// A sink that was never part of a run writes nothing.
//
// The distinction is RunStarted. Without it no document was ever opened, so there
// is nothing to write and inventing one would claim something happened.
//
// AN EMPTY RUN IS DIFFERENT and does produce a document, carrying tests="0" - the
// second half of this test. That is the reverse of the behaviour before RunStarted
// existed, and deliberately so: a missing file is ambiguous, because a
// configuration problem and a run with no tests look identical from CI. R3 one
// level up.
FUNCTION_BLOCK TEST_JUnitReporterWritesNothingWhenNothingRan IMPLEMENTS I_Test
VAR
	Writer : TestJUnitReporter;
	Spy	   : SpyReporter;
	Tally  : TestRunTally;
	Phase  : DINT;
	Scans  : DINT;
	Path : T_MaxString := 'C:\ProgramData\Beckhoff\TwinCAT\3.1\Boot\TestHarnessCoreVerifier_Empty.xml';
	ExpectedCount : UDINT;
	ActualCount	  : UDINT;
END_VAR

METHOD Run : BOOL
VAR_INPUT
	Enable : BOOL;
	Test   : I_TestAssertions;
END_VAR
Scans := Scans + 1;
IF Scans > 2000 THEN
	Test.Fail('the write never finished');
	Run := TRUE;
	RETURN;
END_IF

CASE Phase OF

0:
	Writer.SetPath(Path);
	Writer.AttachErrorSink(Spy);

	// No RunStarted either, so no document is ever opened.
	Tally.SetLabel('nothing');
	Tally.Begin(0);
	Tally.Finish();
	Writer.RunFinished(Status := Tally, TargetInfo := 'the verifier');
	Phase := 1;
	Run	  := FALSE;

1:
	Test.AssertTrue(Writer.IsIdle, 'no write was started');

	ExpectedCount := 0;
	ActualCount	  := Writer.FilesWritten;
	Test.AssertEqual(ExpectedCount, ActualCount, 'nothing was written');

	// Not an error either - an empty run is a legitimate deployment.
	ActualCount := Writer.WriteFailures;
	Test.AssertEqual(ExpectedCount, ActualCount, 'and that is not a failure');

	ActualCount := Spy.FrameworkErrorCalls;
	Test.AssertEqual(ExpectedCount, ActualCount, 'and nothing was reported');

	// Now the same run, announced. An empty run IS an outcome and gets a document.
	Writer.RunStarted(Label := 'nothing', TargetInfo := 'a target');
	Writer.RunFinished(Status := Tally, TargetInfo := 'a target');
	Phase := 2;
	Run	  := FALSE;

2:
	Writer.CyclicLogic();
	IF Writer.IsIdle THEN
		Phase := 3;
	END_IF
	Run := FALSE;

3:
	ExpectedCount := 1;
	ActualCount	  := Writer.FilesWritten;
	Test.AssertEqual(ExpectedCount, ActualCount, 'an announced empty run does write');

	ExpectedCount := 0;
	ActualCount	  := Writer.WriteFailures;
	Test.AssertEqual(ExpectedCount, ActualCount, 'and not as a failure');

	Run := TRUE;

END_CASE
END_METHOD

END_FUNCTION_BLOCK

(* stored: Version 1.1.0.1, ProductVersion 3.1.4026.18
   POU TEST_JUnitReporterWritesNothingWhenNothingRan: Id {650bc756-1aa8-4184-89aa-cf8748b947a9}, SpecialFunc None
   Folder I_Test: Id {743a46e5-6d0b-48e3-b191-60664dedc74d}
   Method Run: Id {20f1a074-cd60-4bf8-b302-bae9f59b2f83} *)
